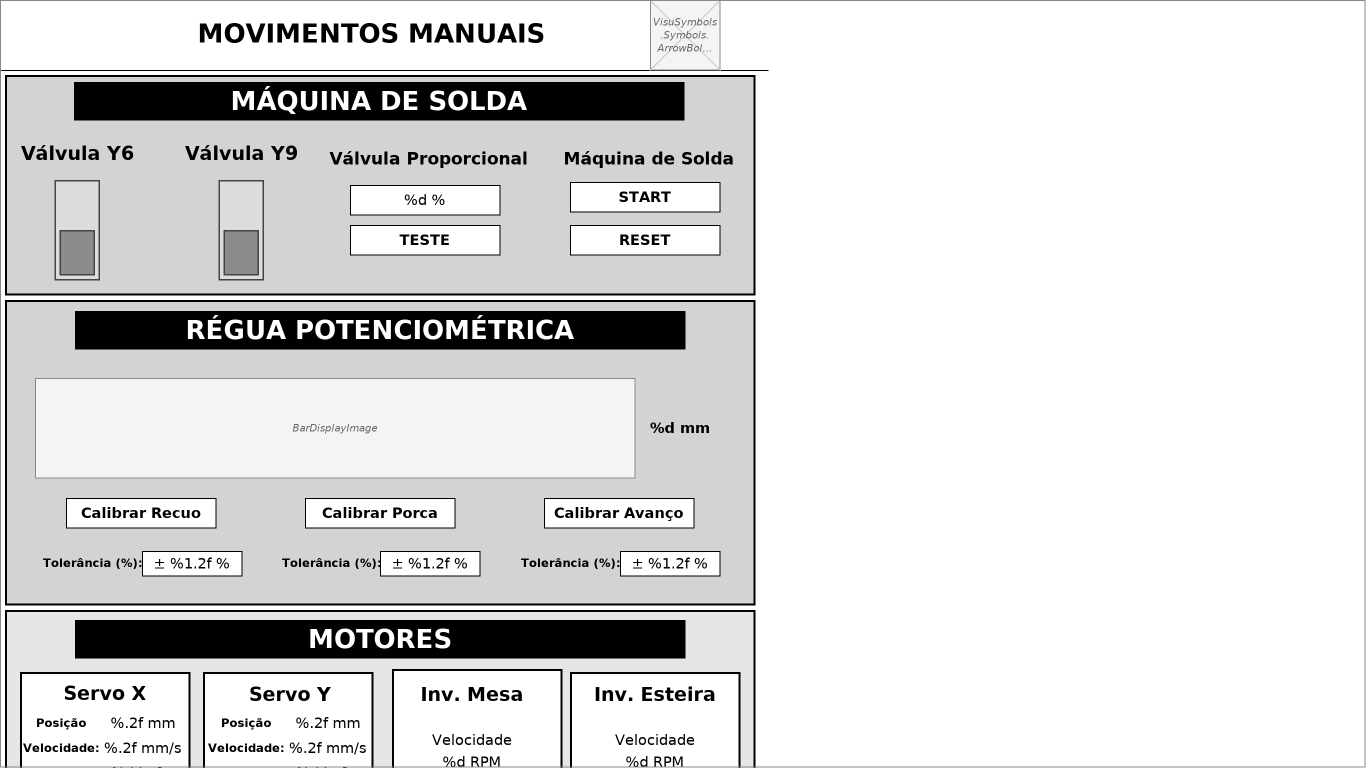
VISUALIZATION Tela_Manual_1  // 1366x768
    Line (0,70) (768,70), input disabled if: NOT MaquinaModoManual
    Line (0,1312) (768,1312)
    Rectangle (584,1340 180x24), "%t[dd/MM/yyyy]"
    Rectangle (584,1316 180x24), "%t[HH:mm:ss]"
    Label (153,7 437x53), "MOVIMENTOS MANUAIS"
    Button (15,1315 175x45), "RECEITAS"
        OnMouseClick: change screen: Tela_Receita
    Button (375,1315 175x45), "MANUTENÇÃO"
        OnMouseClick: change screen: Tela_Manutencao
    RoundedRectangle (5,75 750x220)
    Rectangle (74,82 610x38), "MÁQUINA DE SOLDA", text variable: Recipe_name_Select, input disabled if: NOT MaquinaModoManual
    RoundedRectangle (5,610 750x691), input disabled if: NOT MaquinaModoManual
    Rectangle (75,620 610x38), "MOTORES", text variable: Recipe_name_Select, input disabled if: NOT MaquinaModoManual
    RoundedRectangle (570,672 170x420), input disabled if: NOT MaquinaModoManual
    PushSwitch (625,907 60x60), variable: IhmBt_EsteiraSaida_LigarDesligar, input disabled if: NOT MaquinaModoManual, behaviour: TOGGLE, style: Switch-PushSwitch-Green
    Rectangle (575,681 160x27), "Inv. Esteira", text variable: Recipe_name_Select, input disabled if: NOT MaquinaModoManual
    Rectangle (602,729 106x22), "Velocidade", text variable: Recipe_name_Select, input disabled if: NOT MaquinaModoManual
    Rectangle (602,751 106x22), "%d RPM", text variable: Recipe_name_Select, input disabled if: NOT MaquinaModoManual
    Rectangle (602,879 106x22), "Liga/Desliga", text variable: Recipe_name_Select, input disabled if: NOT MaquinaModoManual
    RotarySwitch (625,803 60x60), variable: IhmBt_EsteiraSaida_Sentido, input disabled if: NOT MaquinaModoManual, behaviour: TOGGLE, style: Switch-RotarySwitch-Gray
    Image (582,823 36x20), input disabled if: NOT MaquinaModoManual, image: VisuSymbols.Symbols.ArrowBoldLeft
    Image (692,823 36x20), input disabled if: NOT MaquinaModoManual, image: VisuSymbols.Symbols.ArrowBoldRight
    RoundedRectangle (392,669 170x420), input disabled if: NOT MaquinaModoManual
    Rectangle (394,681 156x27), "Inv. Mesa", text variable: Recipe_name_Select, input disabled if: NOT MaquinaModoManual
    Rectangle (419,729 106x22), "Velocidade", text variable: Recipe_name_Select, input disabled if: NOT MaquinaModoManual
    Rectangle (419,751 106x22), "%d RPM", text variable: Recipe_name_Select, input disabled if: NOT MaquinaModoManual
    Group (404,803 147x60), input disabled if: NOT MaquinaModoManual
        RotarySwitch (44,0 60x60), variable: IhmBt_MesaIndex_Sentido, behaviour: TOGGLE, style: Switch-RotarySwitch-Gray
        Image (0,20 36x20), image: VisuSymbols.Symbols.ArrowBoldLeft
        Image (111,20 36x20), image: VisuSymbols.Symbols.ArrowBoldRight
    RoundedRectangle (20,672 170x360), input disabled if: NOT MaquinaModoManual
    Rectangle (52,680 106x27), "Servo X", text variable: Recipe_name_Select, input disabled if: NOT MaquinaModoManual
    Rectangle (23,712 77x22), "Posição", input disabled if: NOT MaquinaModoManual
    Rectangle (98,712 90x22), "%.2f mm", text variable: IhmLeit_ServoX_Posicao, input disabled if: NOT MaquinaModoManual
    RoundedRectangle (30,982 150x30), "REFERENCIAR", input disabled if: NOT MaquinaModoManual
        tap IhmBt_ServoX_Referenciar
    RoundedRectangle (30,942 150x30), "POWER ON", input disabled if: NOT MaquinaModoManual
        toggle IhmBt_ServoX_PowerOn
    RoundedRectangle (30,842 150x30), "HOME", colour toggle: NOT Servos.PowerOnServoX, input disabled if: NOT MaquinaModoManual
        tap IhmBt_ServoX_Home
    RoundedRectangle (30,802 150x30), "RESET", input disabled if: NOT MaquinaModoManual
        tap IhmBt_ServoX_Reset
    Image (30,882 50x50), invisible if: NOT IhmBt_ServoX_PowerOn, input disabled if: NOT MaquinaModoManual, image: VisuSymbols.Symbols.ArrowBoldLeft
        OnMouseDown: execute { IhmBt_ServoX_JogBwd := TRUE; }
        OnMouseLeave: execute { IhmBt_ServoX_JogBwd := FALSE; }
        OnMouseUp: execute { IhmBt_ServoX_JogBwd := FALSE; }
    Image (130,882 50x50), invisible if: NOT IhmBt_ServoX_PowerOn, input disabled if: NOT MaquinaModoManual, image: VisuSymbols.Symbols.ArrowBoldRight
        OnMouseDown: execute { IhmBt_ServoX_JogFwd := TRUE; }
        OnMouseLeave: execute { IhmBt_ServoX_JogFwd := FALSE; }
        OnMouseUp: execute { IhmBt_ServoX_JogFwd := FALSE; }
    Rectangle (82,896 45x20), "JOG", invisible if: NOT IhmBt_ServoX_PowerOn, input disabled if: NOT MaquinaModoManual
    Rectangle (23,737 77x22), "Velocidade:", input disabled if: NOT MaquinaModoManual
    Rectangle (98,737 90x22), "%.2f mm/s", text variable: IhmLeit_ServoX_Velocidade, input disabled if: NOT MaquinaModoManual
    Rectangle (23,762 77x22), "Torque:", input disabled if: NOT MaquinaModoManual
    Rectangle (98,762 90x22), "%d kgfm", text variable: IhmLeit_ServoX_Torque, input disabled if: NOT MaquinaModoManual
    RoundedRectangle (203,672 170x360), input disabled if: NOT MaquinaModoManual
    Rectangle (237,681 106x27), "Servo Y", text variable: Recipe_name_Select, input disabled if: NOT MaquinaModoManual
    RoundedRectangle (215,982 150x30), "REFERENCIAR", input disabled if: NOT MaquinaModoManual
        tap IhmBt_ServoY_Referenciar
    RoundedRectangle (215,942 150x30), "POWER ON", input disabled if: NOT MaquinaModoManual
        toggle IhmBt_ServoY_PowerOn
    RoundedRectangle (215,842 150x30), "HOME", colour toggle: NOT Servos.PowerOnServoX, input disabled if: NOT MaquinaModoManual
        tap IhmBt_ServoY_Home
    RoundedRectangle (215,802 150x30), "RESET", input disabled if: NOT MaquinaModoManual
        tap IhmBt_ServoY_Reset
    Image (215,882 50x50), invisible if: NOT IhmBt_ServoY_PowerOn, input disabled if: NOT MaquinaModoManual, image: VisuSymbols.Symbols.ArrowBoldLeft
        OnMouseUp: execute { IhmBt_ServoY_JogBwd := FALSE; }
        OnMouseLeave: execute { IhmBt_ServoY_JogBwd := FALSE; }
        OnMouseDown: execute { IhmBt_ServoY_JogBwd := TRUE; }
    Image (315,882 50x50), invisible if: NOT IhmBt_ServoY_PowerOn, input disabled if: NOT MaquinaModoManual, image: VisuSymbols.Symbols.ArrowBoldRight
        OnMouseUp: execute { IhmBt_ServoY_JogFwd := FALSE; }
        OnMouseLeave: execute { IhmBt_ServoY_JogFwd := FALSE; }
        OnMouseDown: execute { IhmBt_ServoY_JogFwd := TRUE; }
    Rectangle (267,896 45x20), "JOG", text variable: Recipe_name_Select, invisible if: NOT IhmBt_ServoY_PowerOn, input disabled if: NOT MaquinaModoManual
    Rectangle (208,712 77x22), "Posição", input disabled if: NOT MaquinaModoManual
    Rectangle (208,737 77x22), "Velocidade:", input disabled if: NOT MaquinaModoManual
    Rectangle (208,762 77x22), "Torque:", input disabled if: NOT MaquinaModoManual
    Rectangle (283,762 90x22), "%d kgfm", text variable: IhmLeit_ServoY_Torque, input disabled if: NOT MaquinaModoManual
    Rectangle (283,712 90x22), "%.2f mm", text variable: IhmLeit_ServoY_Posicao, input disabled if: NOT MaquinaModoManual
    Rectangle (283,737 90x22), "%.2f mm/s", text variable: IhmLeit_ServoY_Velocidade, input disabled if: NOT MaquinaModoManual
    RoundedRectangle (388,1098 353x125), input disabled if: NOT MaquinaModoManual
    Rectangle (411,1132 130x20), "Frequência (Mesa):", input disabled if: NOT MaquinaModoManual
    Rectangle (584,1132 130x25), "%d Hz", text variable: IhmEscr_MesaIndex_Frequencia, input disabled if: NOT MaquinaModoManual
        OnMouseClick: write the text variable via Default, min 0, max 60
    Rectangle (584,1162 130x25), "%1.2f s", text variable: IhmEscr_MesaIndex_DelayParada, input disabled if: NOT MaquinaModoManual
        OnMouseClick: write the text variable via Default, min 0
    Rectangle (408,1165 130x20), "Delay (Parada)", input disabled if: NOT MaquinaModoManual
    Rectangle (388,1099 353x27), "Ajustes - Inversores", text variable: Recipe_name_Select, input disabled if: NOT MaquinaModoManual
    RoundedRectangle (20,1038 353x185), input disabled if: NOT MaquinaModoManual
    Rectangle (116,1039 160x27), "Ajustes - Servos", text variable: Recipe_name_Select, input disabled if: NOT MaquinaModoManual
    RoundedRectangle (231,1185 50x30), "x100", input disabled if: NOT MaquinaModoManual
        toggle IhmBt_ServoXY_X100
    RoundedRectangle (111,1185 50x30), "x1", input disabled if: NOT MaquinaModoManual
        toggle IhmBt_ServoXY_X1
    RoundedRectangle (171,1185 50x30), "x10", input disabled if: NOT MaquinaModoManual
        toggle IhmBt_ServoXY_X10
    Rectangle (220,1066 130x25), "%d kgf", text variable: IhmEscr_ServoXY_TorqueMax, input disabled if: NOT MaquinaModoManual
        OnMouseClick: write the text variable via Default, min 0, max 300
    Rectangle (44,1069 130x20), "Torque Máximo:", input disabled if: NOT MaquinaModoManual
    Rectangle (220,1095 130x25), "%1.2f s", text variable: IhmEscr_ServoXY_TempoTorqueMax, input disabled if: NOT MaquinaModoManual
        OnMouseClick: write the text variable via Default, min 0, max 300
    Rectangle (43,1098 170x20), "Tempo (Torque Máximo):", input disabled if: NOT MaquinaModoManual
    Rectangle (44,1155 130x20), "Velocidade (Manual):", input disabled if: NOT MaquinaModoManual
    Rectangle (220,1155 130x25), "%d mm/s", text variable: IhmEscr_ServoXY_VelocidadeManual, input disabled if: TRUE
        OnMouseClick: write the text variable via Default, min 0, max 300
    Rectangle (220,1125 130x25), "%d mm/s", text variable: IhmEscr_ServoXY_VelocidadeAuto, input disabled if: NOT MaquinaModoManual
        OnMouseClick: write the text variable via Default, min 0, max 300
    Rectangle (44,1128 130x20), "Velocidade (Auto):", input disabled if: NOT MaquinaModoManual
    Group (404,879 146x192), input disabled if: NOT MaquinaModoManual
        PushSwitch (43,28 60x60), variable: IhmBt_MesaIndex_LigarDesligar, behaviour: TOGGLE, style: Switch-PushSwitch-Green
        Rectangle (20,0 106x22), "Liga/Desliga", text variable: Recipe_name_Select
        PushSwitch (43,132 60x60), variable: IhmBt_MesaIndex_Ciclo, behaviour: TAP, style: Switch-PushSwitch-Green
        Rectangle (0,104 146x22), "Revolução", text variable: Recipe_name_Select
    Image (650,0 70x70), image: VisuSymbols.Symbols.ArrowBoldRight
        OnMouseClick: change screen: Tela_Manual_2
    Image (686,1148 0x1), input disabled if: NOT MaquinaModoManual, image: ImagePool.bt_REFRESH
    Rectangle (584,1192 130x25), "%d Hz", text variable: IhmEscr_EsteiraSaida_Frequencia, input disabled if: NOT MaquinaModoManual
        OnMouseClick: write the text variable via Default, min 0, max 300
    Rectangle (408,1195 130x20), "Frequência (Esteira):", input disabled if: NOT MaquinaModoManual
    Button (195,1315 175x45), "PRODUÇÃO"
        OnMouseClick: change screen: Tela_Producao
    Button (260,1235 240x60), "MODO: %s", text variable: IhmBt_ManualAuto_Text, colour toggle: IhmBt_ManualAuto_Color
        toggle IhmBt_ManualAuto
    Group (20,140 279x140), input disabled if: NOT MaquinaModoManual
        Rectangle (0,0 115x27), "Válvula Y6", text variable: Recipe_name_Select, input disabled if: MaquinaModoAuto
        DipSwitch (7,40 100x100), variable: IhmBt_Y6_Ligar, input disabled if: MaquinaModoAuto, behaviour: TOGGLE, style: Switch-DipSwitch-Gray
        Rectangle (164,0 115x27), "Válvula Y9", text variable: Recipe_name_Select, input disabled if: MaquinaModoAuto
        DipSwitch (171,40 100x100), variable: IhmBt_Y9_Ligar, input disabled if: MaquinaModoAuto, behaviour: TOGGLE, style: Switch-DipSwitch-Gray
    Rectangle (319,145 220x27), "Válvula Proporcional", text variable: Recipe_name_Select, input disabled if: NOT MaquinaModoManual
    RoundedRectangle (350,225 150x30), "TESTE", colour toggle: NOT Servos.PowerOnServoX, input disabled if: NOT MaquinaModoManual
        tap IhmBt_VP_Teste
    Rectangle (350,185 150x30), "%d %", text variable: IhmEscr_ValvulaProporcional, input disabled if: NOT MaquinaModoManual
        OnMouseClick: write the text variable via Default, min 0, max 100
    Rectangle (539,145 220x27), "Máquina de Solda", text variable: Recipe_name_Select, input disabled if: NOT MaquinaModoManual
    RoundedRectangle (570,225 150x30), "RESET", colour toggle: NOT Servos.PowerOnServoX, input disabled if: NOT MaquinaModoManual
        tap IhmBt_MaquinaSolda_Reset
    RoundedRectangle (570,182 150x30), "START", colour toggle: NOT Servos.PowerOnServoX, input disabled if: NOT MaquinaModoManual
        toggle IhmBt_MaquinaSolda_Start
    RoundedRectangle (5,300 750x305)
    Rectangle (75,311 610x38), "RÉGUA POTENCIOMÉTRICA", text variable: Recipe_name_Select, input disabled if: NOT MaquinaModoManual
    Group (35,378 690x198)
        RoundedRectangle (31,120 150x30), "Calibrar Recuo", input disabled if: NOT MaquinaModoManual
            tap IhmBt_ReguaPotenciometrica_CalibrarRecuo
        Rectangle (5,175 100x20), "Tolerância (%):", input disabled if: NOT MaquinaModoManual
        BarDisplayImage (0,0 600x100), value: ReguaPotenciometricaPosicao, style: BarDisplayImage-Gray, scale format: %.1f, scale 0..100
            p518627256: mm
        Rectangle (600,39 90x22), "%d mm", text variable: ReguaPotenciometricaPosicao, input disabled if: TRUE
        Rectangle (244,175 100x20), "Tolerância (%):", input disabled if: NOT MaquinaModoManual
        RoundedRectangle (270,120 150x30), "Calibrar Porca", input disabled if: NOT MaquinaModoManual
            tap IhmBt_ReguaPotenciometrica_CalibrarPorca
        RoundedRectangle (509,120 150x30), "Calibrar Avanço", input disabled if: NOT MaquinaModoManual
            tap IhmBt_ReguaPotenciometrica_CalibrarAvanco
        Rectangle (483,175 100x20), "Tolerância (%):", input disabled if: NOT MaquinaModoManual
        Rectangle (107,173 100x25), "± %1.2f %", text variable: IhmEscr_ReguaPotenciometrica_ToleranciaRecuo, input disabled if: NOT MaquinaModoManual
            OnMouseClick: write the text variable via Default, min 0, max 100
        Rectangle (345,173 100x25), "± %1.2f %", text variable: IhmEscr_ReguaPotenciometrica_ToleranciaPorca, input disabled if: NOT MaquinaModoManual
            OnMouseClick: write the text variable via Default, min 0, max 100
        Rectangle (585,173 100x25), "± %1.2f %", text variable: IhmEscr_ReguaPotenciometrica_ToleranciaAvanco, input disabled if: NOT MaquinaModoManual
            OnMouseClick: write the text variable via Default, min 0, max 100
END_VISUALIZATION

(* stored: Version 1.1.0.1, ProductVersion 3.1.4024.11
   Visu Tela_Manual_1: Id {ea23301c-36e6-447b-8701-8b56ea603908} *)
